SUBAPPLICATION AUI_FIELDBUS_UINT_TO_AR (* AUI-Rohwert (TECU UINT) -> AR, NOT_AVAILABLE/ERROR_INDI-gefiltert (VALID_SIGNAL_W/ERROR_INDI_W/NOT_AVAILABLE_W, FIELDBUS_SIGNAL.gcf), unskaliert (SCALE=1.0/OFFSET=0 fest). *)
  (* Standard: 61499-2; Description: Copyright (c) 2026 Meisterschulen am Ostbahnhof This program and the accompanying materials are made available under the terms of the Eclipse Public License 2.0 which is available at https://www.eclipse.org/legal/epl-2.0/ SPDX-License-Identifier: EPL-2.0 *)
  (* Version 1.1, 2026-09-16, Franz Höpfinger, Meisterschulen am Ostbahnhof, Nach MyLib_AX-1.0.0::sys verschoben (Franz) - generischer Baustein, gehoert nicht in den TECU-spezifischen Ordner. *)
  (* Version 1.0, 2026-09-16, Franz Höpfinger, Meisterschulen am Ostbahnhof, Herausgeloest (Franz: 'AUI_FIELDBUS_UINT_TO_SIGNAL_SCALED mit SCALE 1 und OFFSET 0 kann auch eine SUB sein') - in TECU_RPTO/TECU_FPTO/TECU_COGSOG/TECU_GBSD/TECU_WBSD/TECU_VDS/TECU_FHS/TECU_RHS wurde SCALE=1.0/OFFSET=0 bisher jedes Mal einzeln parametriert. *)
  PACKAGE MyLib::sys;
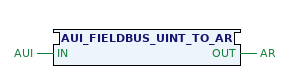
  SOCKETS
    IN : adapter::types::unidirectional::AUI; (* TECU-Rohwert *)
  END_SOCKETS
  PLUGS
    OUT : adapter::types::unidirectional::AR; (* 0.0 bei NOT_AVAILABLE/ERROR_INDI, sonst IN unskaliert *)
  END_PLUGS
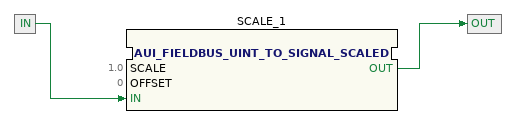
  FBS
    SCALE_1 : logiBUS::signalprocessing::fieldbus::AUI_FIELDBUS_UINT_TO_SIGNAL_SCALED(SCALE := 1.0, OFFSET := 0);
  END_FBS
  ADAPTER_CONNECTIONS
    IN TO SCALE_1.IN;
    SCALE_1.OUT TO OUT;
  END_CONNECTIONS
END_SUBAPPLICATION
